FUNCTION_BLOCK Technology EXTENDS TcoCore.TcoContext
VAR
	_ST001 : ST001(THIS^);
END_VAR

(*~
	<docu>
		<summary>
			Main method of the TcoContext. This is the entry point of any control logic that belongs to this context. 
			The call of this method is ensured by calling the <c>InstanceName.Run()</c> method, and it must not be called explicitly.
			This method is abstract, and it must be overridden in derived block.
		</summary>
	</docu>
~*)
METHOD PROTECTED  Main
_ST001();
END_METHOD

END_FUNCTION_BLOCK

(* stored: Version 1.1.0.1, ProductVersion 3.1.4024.9
   POU Technology: Id {f5d907bb-c69e-0cce-3445-38466ba70424}, SpecialFunc None
   Method Main: Id {c95e53db-9583-06d0-14c2-b6db009198f1} *)
